TYPE ST_Timers :
STRUCT
	
	nStation1TimeOut				: DINT			:= 10;
	nStation2TimeOut				: DINT			:= 10;
	nStation3TimeOut				: DINT			:= 10;

END_STRUCT
END_TYPE

(* stored: Version 1.1.0.1, ProductVersion 3.1.4024.13
   DUT ST_Timers: Id {9021a1a9-aac4-4fae-9346-03545d78fd35} *)
